# EPICS autosave request: iocBoot/gmca_23b_ioc1/dbSave/bluiceScreening.req
$(P)MountNextXtal
$(P)CenterXtal
$(P)Pause4ctrng
$(P)TakeImage0
$(P)TakeImage45
$(P)TakeImage90
$(P)AngleImage0
$(P)AngleImage45
$(P)AngleImage90
$(P)Pause4collect
$(P)RunWebIce
$(P)CurrentTask

$(P)spreadsheetStatus
$(P)spreadsheetDir
$(P)spreadsheetDir0
$(P)spreadsheetDir1
$(P)spreadsheetDir2
$(P)spreadsheetFile

$(P)ScreeningStatus
$(P)spreadsheetSelected
$(P)spreadsheetScreened

$(P)directory
$(P)directory0
$(P)directory1
$(P)directory2
